              if(rq_write_lbl_request[index]):
                  if(is_ack(rq_comm_set_var("LBL", rq_write_lbl[index], socket))):
                      rq_write_lbl_previous[index] = rq_write_lbl[index]
                      rq_write_lbl_request[index] = False
                  end
              end

              if(rq_write_lgn_request[index]):
                  if(is_ack(rq_comm_set_var("LGN", rq_write_lgn[index], socket))):
                      rq_write_lgn_previous[index] = rq_write_lgn[index]
                      rq_write_lgn_request[index] = False
                  end
              end

              if(rq_write_msc_request[index]):
                  if(is_ack(rq_comm_set_var("MSC", rq_write_msc[index], socket))):
                      rq_write_msc_previous[index] = rq_write_msc[index]
                      rq_write_msc_request[index] = False
                  end
              end

              if(rq_write_mod_request[index]):
                  if(is_ack(rq_comm_set_var("MOD", rq_write_mod[index], socket))):
                      rq_write_mod_previous[index] = rq_write_mod[index]
                      rq_write_mod_request[index] = False
                  end
              end
          end
          index = index + 1
      end
  end

  def rq_activate(gripper_socket="1"):
      if (not rq_is_gripper_activated(gripper_socket)):
          rq_reset(gripper_socket)

          while(not rq_get_var("ACT", 1, gripper_socket) == 0 or not rq_get_var("STA", 1, gripper_socket) == 0):
              rq_reset(gripper_socket)
              sync()
          end

          rq_set_var("ACT",1, gripper_socket)
      end
  end

  def rq_activate_and_wait(gripper_socket="1"):
      if (not rq_is_gripper_activated(gripper_socket)):
          rq_activate(gripper_socket)
          sleep(1.0)

          while(not rq_get_var("ACT", 1, gripper_socket) == 1 or not rq_get_var("STA", 1, gripper_socket) == 3):
              sleep(0.1)
          end

          sleep(0.5)
      end
  end

  def rq_activate_all_grippers(reset=False):
      if(gripper_connected[0]):
          rq_reset_and_activate("1", reset)
      end

      if(gripper_connected[1]):
          rq_reset_and_activate("2", reset)
      end

      if(gripper_connected[2]):
          rq_reset_and_activate("3", reset)
      end

      if(gripper_connected[3]):
          rq_reset_and_activate("4", reset)
      end
  end

  def rq_reset_and_activate(gripper_socket="1", reset=False):
      if(reset):
          rq_reset(gripper_socket)
          rq_activate_and_wait(gripper_socket)
      elif(not rq_is_gripper_activated(gripper_socket)):
          rq_activate_and_wait(gripper_socket)
      end
  end

  def rq_reset(gripper_socket="1"):
      rq_set_var("ACT", 0, gripper_socket)
      rq_set_var("ATR", 0, gripper_socket)

      while(not rq_get_var("ACT", 1, gripper_socket) == 0 or not rq_get_var("STA", 1, gripper_socket) == 0):
          rq_set_var("ACT", 0, gripper_socket)
          rq_set_var("ATR", 0, gripper_socket)
          sync()
      end

      sleep(0.5)
  end

  def rq_auto_release_open_and_wait(gripper_socket="1"):
      rq_set_var("ATR",0, gripper_socket)
      rq_set_var("ARD",0, gripper_socket)
      rq_set_var("ACT",1, gripper_socket)
      sleep(0.1)
      rq_set_var("ATR",1, gripper_socket)

      rq_wait_autorelease_completed(gripper_socket)
  end

  def rq_auto_release_close_and_wait(gripper_socket="1"):
      rq_set_var("ATR",0, gripper_socket)
      rq_set_var("ARD",1, gripper_socket)
      rq_set_var("ACT",1, gripper_socket)
      sleep(0.1)
      rq_set_var("ATR",1, gripper_socket)

      rq_wait_autorelease_completed(gripper_socket)
  end

  def rq_wait_autorelease_completed(gripper_socket="1"):
      remainingRetries = 20
      gFLT = rq_get_var("FLT", 2, gripper_socket)

      while(not is_FLT_autorelease_in_progress(gFLT) and remainingRetries > 0):
          remainingRetries = remainingRetries - 1
          gFLT = rq_get_var("FLT", 2, gripper_socket)
          sleep(0.1)
      end

      remainingRetries = 100
      gFLT = rq_get_var("FLT", 2, gripper_socket)

      while(not is_FLT_autorelease_completed(gFLT) and remainingRetries > 0):
          remainingRetries = remainingRetries - 1
          gFLT = rq_get_var("FLT", 2, gripper_socket)
          sleep(0.1)
      end
  end

  def rq_set_force(force, gripper_socket="1"):
      force = floor(scale(force, [0, 255], [0.0, 255.0]))
      rq_set_var("FOR", force, gripper_socket)
  end

  def rq_set_speed(speed, gripper_socket="1"):
      speed = floor(scale(speed, [0, 255], [0.0, 255.0]))
      rq_set_var("SPE", speed, gripper_socket)
  end

  def rq_open(gripper_socket="1"):
      rq_move(0, gripper_socket)
  end

  def rq_close(gripper_socket="1"):
      rq_move(255, gripper_socket)
  end

  def rq_open_and_wait(gripper_socket="1"):
      rq_move_and_wait(0, gripper_socket)
  end

  def rq_close_and_wait(gripper_socket="1"):
      rq_move_and_wait(255, gripper_socket)
  end

  def rq_move(pos, gripper_socket="1"):
      rq_set_pos(pos, gripper_socket)
      rq_go_to(gripper_socket)
  end

  def rq_move_and_wait(pos, gripper_socket="1"):
      rq_move(pos, gripper_socket)

      while (not rq_is_motion_complete(gripper_socket)):
          # wait for motion completed
          sync()
      end
  end

  def rq_wait_for_pos_request(pos, gripper_socket="1"):
      gPRE = rq_get_var("PRE", 3, gripper_socket)

      while (gPRE != pos):
          rq_set_var("POS", pos, gripper_socket)
          sync()
          gPRE = rq_get_var("PRE", 3, gripper_socket)
      end
  end

  def rq_wait_pos_spe_for_request(pos, speed, force, gripper_socket="1"):
      gPRE = rq_get_var("PRE", 3, gripper_socket)

      while (gPRE != pos):
          rq_set_pos_spe_for_var(pos, speed, force, gripper_socket)
          sync()
          gPRE = rq_get_var("PRE", 3, gripper_socket)
      end
  end

  def rq_wait_for_pos(pos, gripper_socket="1"):
      rq_wait_for_pos_request(pos, gripper_socket)

      # Wait for the gripper motion to complete
      while (not rq_is_motion_complete(gripper_socket)):
          # wait for motion completed
          sync()
          rq_set_var("GTO", 1, gripper_socket)
      end
  end

  def rq_wait(gripper_socket="1"):
      # Wait for the gripper motion to complete
      while (not rq_is_motion_complete(gripper_socket)):
          sync()
          # The following patch is for Robotiq's Camera issue when communication is lost, but not the activation
          # the communication driver reset the GTO bit
          rq_set_var("GTO", 1, gripper_socket)
      end
  end

  def rq_wait_for_object_detected(gripper_socket="1"):
      # Wait the object detection
      while (not rq_is_object_detected(gripper_socket)):
          sync()
      end
  end

  # set the position
  def rq_set_pos(pos, gripper_socket="1"):
      pos = floor(scale(pos, [0, 255], [0.0, 255.0]))
      rq_set_var("POS", pos, gripper_socket)
      rq_wait_for_pos_request(pos, gripper_socket)
  end

  def rq_set_pos_spd_for(pos, speed, force, gripper_socket="1"):
      pos = floor(scale(pos, [0, 255], [0.0, 255.0]))
      speed = floor(scale(speed, [0, 255], [0.0, 255.0]))
      force = floor(scale(force, [0, 255], [0.0, 255.0]))

      rq_set_pos_spe_for_var(pos, speed, force, gripper_socket)
  end

  def rq_set_gripper_max_current_mA(current_mA, gripper_socket="1"):
      current = floor(current_mA / 10)

      rq_set_var("MSC", current, gripper_socket)
      current_read = rq_get_var("MSC", 1, gripper_socket)

      while(current_read != current):
          rq_set_var("MSC", current, gripper_socket)
          current_read = rq_get_var("MSC", 1, gripper_socket)
      end
  end

  def rq_set_gripper_mode(mode, gripper_socket="1"):
      rq_set_var("MOD", mode, gripper_socket)
  end

  def rq_set_gripper_max_cur(current_mA, gripper_socket="1"):
      rq_set_gripper_max_current_mA(current_mA, gripper_socket)
  end

  def rq_get_gripper_max_current_mA(gripper_socket="1"):
      current = rq_get_var("MSC", 1, gripper_socket)

      if(current == -1):
          current_mA = current
      else:
          current_mA = current * 10
      end

      return current_mA
  end

  def rq_get_gripper_max_cur(gripper_socket="1"):
      return rq_get_gripper_max_current_mA(gripper_socket)
  end

  def rq_set_max_current_for_all_grippers():
      current_mA = rq_get_max_current_mA()

      if(gripper_connected[0]):
          rq_set_gripper_max_current_mA(current_mA, "1")
      end

      if(gripper_connected[1]):
          rq_set_gripper_max_current_mA(current_mA, "2")
      end

      if(gripper_connected[2]):
          rq_set_gripper_max_current_mA(current_mA, "3")
      end

      if(gripper_connected[3]):
          rq_set_gripper_max_current_mA(current_mA, "4")
      end
  end

  def rq_get_max_current_mA():
      max_current_mA = 0

      if(rq_current_limit_enabled):
          nb_connected_grippers = rq_get_nb_connected_grippers()

          if(nb_connected_grippers == 1):
              max_current_mA = 600
          elif(nb_connected_grippers > 1):
              max_current_mA = 450
          end
      else:

      end

      return max_current_mA
  end

  def rq_get_nb_connected_grippers():
      nb_connected_grippers = 0

      if(gripper_connected[0]):
          nb_connected_grippers = nb_connected_grippers + 1
      end

      if(gripper_connected[1]):
          nb_connected_grippers = nb_connected_grippers + 1
      end

      if(gripper_connected[2]):
          nb_connected_grippers = nb_connected_grippers + 1
      end

      if(gripper_connected[3]):
          nb_connected_grippers = nb_connected_grippers + 1
      end

      return nb_connected_grippers
  end

  def rq_list_of_bytes_to_value(list_of_bytes):
      value = -1

      # response list length
      if (list_of_bytes[0] == 1):
          value = list_of_bytes[1] - 48
      elif (list_of_bytes[0] == 2):
          value = (list_of_bytes[1] - 48) * 10 + (list_of_bytes[2] - 48)
      elif (list_of_bytes[0] == 3):
          value = (list_of_bytes[1] - 48) * 100 + (list_of_bytes[2] - 48) * 10 + (list_of_bytes[3] - 48)
      end

      return value
  end

  def rq_is_motion_complete(gripper_socket="1"):
      gOBJ = rq_get_var("OBJ", 1, gripper_socket)
      sync()
      return is_OBJ_gripper_at_position(gOBJ) or is_OBJ_object_detected(gOBJ)
  end

  def rq_is_gripper_activated(gripper_socket="1"):
      gSTA = rq_get_var("STA", 1, gripper_socket)
      sync()
      return is_STA_gripper_activated(gSTA)
  end

  def rq_is_object_detected(gripper_socket="1"):
      gOBJ = rq_get_var("OBJ", 1, gripper_socket)
      sync()
      return is_OBJ_object_detected(gOBJ)
  end

  def rq_current_pos(gripper_socket="1"):
      gPOS = rq_get_var("POS", 1, gripper_socket)
      sync()
      return gPOS
  end

  def rq_motor_current(gripper_socket="1"):
      rq_current = rq_get_var("COU", 1, gripper_socket)
      sync()
      return rq_current * 10
  end

  def rq_print_connected_grippers():
      if(gripper_connected[0]):
          textmsg("Gripper 1 : ", "connected and socket open.")
      end

      if (gripper_connected[1]):
          textmsg("Gripper 2 : ", "connected and socket open.")
      end

      if (gripper_connected[2]):
          textmsg("Gripper 3 : ", "connected and socket open.")
      end

      if (gripper_connected[3]):
          textmsg("Gripper 4 : ", "connected and socket open.")
      end
  end

  def rq_print_gripper_fault_code(gripper_socket="1"):
      gFLT = rq_get_var("FLT", 2, gripper_socket)

      if(is_FLT_no_fault(gFLT)):
          textmsg("Gripper Fault : ", "No Fault (0x00)")
      elif (is_FLT_action_delayed(gFLT)):
          textmsg("Gripper Fault : ", "Priority Fault: Action delayed, initialization must be completed prior to action (0x05)")
      elif (is_FLT_not_activated(gFLT)):
          textmsg("Gripper Fault : ", "Priority Fault: The activation must be set prior to action (0x07)")
      elif (is_FLT_autorelease_in_progress(gFLT)):
          textmsg("Gripper Fault : ", "Minor Fault: Automatic release in progress (0x0B)")
      elif (is_FLT_overcurrent(gFLT)):
          textmsg("Gripper Fault : ", "Minor Fault: Overcurrent protection triggered (0x0E)")
      elif (is_FLT_autorelease_completed(gFLT)):
          textmsg("Gripper Fault : ", "Major Fault: Automatic release completed (0x0F)")
      else:
          textmsg("Gripper Fault : ", "Unknown Fault")
      end
  end

  def rq_print_gripper_num_cycles(gripper_socket="1"):
      num_cycles = rq_get_var("NCY", 1, gripper_socket)

      if(num_cycles == -1):
          textmsg("Gripper Cycle Number : ", "Number of cycles is unreachable.")
      else:
          textmsg("Gripper Cycle Number : ", num_cycles)
      end
  end

  def rq_print_gripper_driver_state(gripper_socket="1"):
      driver_state = rq_get_var("DST", 1, gripper_socket)

      if(driver_state == 0):
          textmsg("Gripper Driver State : ", "RQ_STATE_INIT")
      elif(driver_state == 1):
          textmsg("Gripper Driver State : ", "RQ_STATE_LISTEN")
      elif(driver_state == 2):
          textmsg("Gripper Driver State : ", "RQ_STATE_READ_INFO")
      elif(driver_state == 3):
          textmsg("Gripper Driver State : ", "RQ_STATE_ACTIVATION")
      else:
          textmsg("Gripper Driver State : ", "RQ_STATE_RUN")
      end
  end

  def rq_print_gripper_serial_number(gripper_socket="1"):
      serial_number = rq_get_var_string("SNU", 1, gripper_socket)
      textmsg("Gripper Serial Number : ", serial_number)
  end

  def rq_print_gripper_firmware_version(gripper_socket="1"):
      firmware_version = rq_get_var_string("FWV", 1, gripper_socket)
      textmsg("Gripper Firmware Version : ", firmware_version)
  end

  def rq_print_gripper_driver_version(gripper_socket="1"):
      driver_version = rq_get_var_string("VER", 1, gripper_socket)
      textmsg("Gripper Driver Version : ", driver_version)
  end

  def rq_print_gripper_connection_state(gripper_socket="1"):
      connection_state = rq_get_var("PCO", 1, gripper_socket)

      if (connection_state == 0):
          textmsg("Gripper Connection State : ", "No connection problem detected")
      else:
          textmsg("Gripper Connection State : ", "Connection problem detected")
      end
  end

  # Returns True if list_of_bytes is [3, 'a', 'c', 'k']
  def is_ack(list_of_bytes):

      # list length is not 3
      if (list_of_bytes[0] != 3):
          return False
      end

      # first byte not is 'a'?
      if (list_of_bytes[1] != 97):
          return False
      end

      # first byte not is 'c'?
      if (list_of_bytes[2] != 99):
          return False
      end

      # first byte not is 'k'?
      if (list_of_bytes[3] != 107):
          return False
      end

      return True
  end

  # Returns True if list_of_bytes is not [3, 'a', 'c', 'k']
  def is_not_ack(list_of_bytes):
      if (is_ack(list_of_bytes)):
          return False
      else:
          return True
      end
  end

  def is_STA_gripper_activated (gSTA):
      if (gSTA == 3):
          return True
      end

      return False
  end

  def is_OBJ_object_detected (gOBJ):
      if (gOBJ == 1 or gOBJ == 2):
          return True
      end

      return False
  end

  def is_OBJ_gripper_at_position (gOBJ):
      if (gOBJ == 3):
          return True
      end

      return False
  end

  def is_not_OBJ_gripper_at_position (gOBJ):
      if (is_OBJ_gripper_at_position(gOBJ)):
          return False
      else:
          return True
      end
  end

  #### GTO Section ####
  def rq_stop(gripper_socket="1"):
      rq_set_var("GTO", 0, gripper_socket)
  end

  def rq_set_GTO_and_wait(value, gripper_socket="1"):
      rq_set_var("GTO" ,value, gripper_socket)
      while(not is_GTO(value, rq_get_var("GTO", 1, gripper_socket))):
        sync()
      end
  end

  def rq_go_to(gripper_socket="1"):
      rq_set_var("GTO", 1, gripper_socket)
  end


  def is_GTO(goto_value, rGTO):
      return rGTO == goto_value
  end
  #### GTO Section ####

  def is_FLT_no_fault(gFLT):
      return gFLT == 0
  end

  def is_FLT_warning(gFLT):
      return gFLT >= 1 and gFLT <= 7
  end

  def is_FLT_faulted(gFLT):
      return gFLT >= 8
  end

  def is_FLT_action_delayed(gFLT):
      return gFLT == 5
  end

  def is_FLT_not_activated(gFLT):
      return gFLT == 7
  end

  def is_FLT_autorelease_in_progress(gFLT):
      return gFLT == 11
  end

  def is_FLT_overcurrent(gFLT):
      return gFLT == 14
  end

  def is_FLT_autorelease_completed(gFLT):
      return gFLT == 15
  end

  def rq_set_var(var_name, var_value, gripper_socket="1"):
      index = rq_socket_to_index(gripper_socket)

      enter_critical

      if (var_name == "ACT"):
          rq_write_act[index] = var_value
          rq_write_act_request[index] = True
      elif (var_name == "GTO"):
          rq_write_gto[index] = var_value
          rq_write_gto_request[index] = True
      elif (var_name == "ATR"):
          rq_write_atr[index] = var_value
          rq_write_atr_request[index] = True
      elif (var_name == "ARD"):
          rq_write_ard[index] = var_value
          rq_write_ard_request[index] = True
      elif (var_name == "FOR"):
          rq_write_for[index] = var_value
          rq_write_pos_request[index] = True
      elif (var_name == "SPE"):
          rq_write_spe[index] = var_value
          rq_write_pos_request[index] = True
      elif (var_name == "POS"):
          rq_write_pos[index] = var_value
          rq_write_pos_request[index] = True
      elif (var_name == "LBP"):
          rq_write_lbp[index] = var_value
          rq_write_lbp_request[index] = True
      elif (var_name == "LRD"):
          rq_write_lrd[index] = var_value
          rq_write_lrd_request[index] = True
      elif (var_name == "LBL"):
          rq_write_lbl[index] = var_value
          rq_write_lbl_request[index] = True
      elif (var_name == "LGN"):
          rq_write_lgn[index] = var_value
          rq_write_lgn_request[index] = True
      elif (var_name == "MSC"):
          rq_write_msc[index] = var_value
          rq_write_msc_request[index] = True
      elif (var_name == "MOD"):
          rq_write_mod[index] = var_value
          rq_write_mod_request[index] = True
      end

      exit_critical

      if (var_name == "ACT"):
          while(rq_write_act_request[index]):
              sync()
          end
      elif (var_name == "GTO"):
          while(rq_write_gto_request[index]):
              sync()
          end
      elif (var_name == "ATR"):
          while(rq_write_atr_request[index]):
              sync()
          end
      elif (var_name == "ARD"):
          while(rq_write_ard_request[index]):
              sync()
          end
      elif (var_name == "FOR"):
          while(rq_write_pos_request[index]):
              sync()
          end
      elif (var_name == "SPE"):
          while(rq_write_pos_request[index]):
              sync()
          end
      elif (var_name == "POS"):
          while(rq_write_pos_request[index]):
              sync()
          end
      elif (var_name == "LBP"):
          while(rq_write_lbp_request[index]):
              sync()
          end
      elif (var_name == "LRD"):
          while(rq_write_lrd_request[index]):
              sync()
          end
      elif (var_name == "LBL"):
          while(rq_write_lbl_request[index]):
              sync()
          end
      elif (var_name == "LGN"):
          while(rq_write_lgn_request[index]):
              sync()
          end
      elif (var_name == "MSC"):
          while(rq_write_msc_request[index]):
              sync()
          end
      elif (var_name == "MOD"):
          while(rq_write_mod_request[index]):
              sync()
          end
      end
  end

  def rq_set_pos_spe_for_var(pos, speed, force, gripper_socket="1"):
      index = rq_socket_to_index(gripper_socket)

      enter_critical

      rq_write_for[index] = force
      rq_write_spe[index] = speed
      rq_write_pos[index] = pos
      rq_write_pos_request[index] = True

      exit_critical
  end

  def rq_get_var(var_name, nbr_bytes, gripper_socket="1"):
      index = rq_socket_to_index(gripper_socket)
      var_value = -1

      if (var_name == "ACT"):
          enter_critical
          rq_read_act_req[index] = True
          exit_critical
          while(rq_read_act_req[index]):
              sync()
          end
          var_value = rq_read_act[index]

      elif (var_name == "GTO"):
          enter_critical
          rq_read_gto_req[index] = True
          exit_critical
          while(rq_read_gto_req[index]):
              sync()
          end
          var_value = rq_read_gto[index]

      elif (var_name == "FOR"):
          enter_critical
          rq_read_for_req[index] = True
          exit_critical
          while(rq_read_for_req[index]):
              sync()
          end
          var_value = rq_read_for[index]

      elif (var_name == "SPE"):
          enter_critical
          rq_read_spe_req[index] = True
          exit_critical
          while(rq_read_spe_req[index]):
              sync()
          end
          var_value = rq_read_spe[index]

      elif (var_name == "OBJ"):
          enter_critical
          rq_read_obj_req[index] = True
          exit_critical
          while(rq_read_obj_req[index]):
              sync()
          end
          var_value = rq_read_obj[index]

      elif (var_name == "STA"):
          enter_critical
          rq_read_sta_req[index] = True
          exit_critical
          while(rq_read_sta_req[index]):
              sync()
          end
          var_value = rq_read_sta[index]

      elif (var_name == "FLT"):
          enter_critical
          rq_read_flt_req[index] = True
          exit_critical
          while(rq_read_flt_req[index]):
              sync()
          end
          var_value = rq_read_flt[index]

      elif (var_name == "POS"):
          enter_critical
          rq_read_pos_req[index] = True
          exit_critical
          while(rq_read_pos_req[index]):
              sync()
          end
          var_value = rq_read_pos[index]

      elif (var_name == "PRE"):
          enter_critical
          rq_read_pre_req[index] = True
          exit_critical
          while(rq_read_pre_req[index]):
              sync()
          end
          var_value = rq_read_pre[index]

      elif (var_name == "LBP"):
          enter_critical
          rq_read_lbp_req[index] = True
          exit_critical
          while(rq_read_lbp_req[index]):
              sync()
          end
          var_value = rq_read_lbp[index]

      elif (var_name == "LRD"):
          enter_critical
          rq_read_lrd_req[index] = True
          exit_critical
          while(rq_read_lrd_req[index]):
              sync()
          end
          var_value = rq_read_lrd[index]

      elif (var_name == "LBL"):
          enter_critical
          rq_read_lbl_req[index] = True
          exit_critical
          while(rq_read_lbl_req[index]):
              sync()
          end
          var_value = rq_read_lbl[index]

      elif (var_name == "LGN"):
          enter_critical
          rq_read_lgn_req[index] = True
          exit_critical
          while(rq_read_lgn_req[index]):
              sync()
          end
          var_value = rq_read_lgn[index]

      elif (var_name == "MSC"):
          enter_critical
          rq_read_msc_req[index] = True
          exit_critical
          while(rq_read_msc_req[index]):
              sync()
          end
          var_value = rq_read_msc[index]

      elif (var_name == "MOD"):
          enter_critical
          rq_read_mod_req[index] = True
          exit_critical
          while(rq_read_mod_req[index]):
              sync()
          end
          var_value = rq_read_mod[index]

      elif (var_name == "NCY"):
          enter_critical
          rq_read_ncy_req[index] = True
          exit_critical
          while(rq_read_ncy_req[index]):
              sync()
          end
          var_value = rq_read_ncy[index]

      elif (var_name == "PCO"):
          enter_critical
          rq_read_pco_req[index] = True
          exit_critical
          while(rq_read_pco_req[index]):
              sync()
          end
          var_value = rq_read_pco[index]

      elif (var_name == "DST"):
          enter_critical
          rq_read_dst_req[index] = True
          exit_critical
          while(rq_read_dst_req[index]):
              sync()
          end
          var_value = rq_read_dst[index]

      end

      return var_value
  end

  def rq_get_var_string(var_name, nbr_bytes, gripper_socket="1"):
      index = rq_socket_to_index(gripper_socket)
      var_value = ""

      enter_critical

      if (var_name == "SNU"):
          if(gripper_socket == "1"):
              var_value = rq_read_snu_1
          elif(gripper_socket == "2"):
              var_value = rq_read_snu_2
          elif(gripper_socket == "3"):
              var_value = rq_read_snu_3
          elif(gripper_socket == "4"):
              var_value = rq_read_snu_4
          end
      elif (var_name == "FWV"):
          if(gripper_socket == "1"):
              var_value = rq_read_fwv_1
          elif(gripper_socket == "2"):
              var_value = rq_read_fwv_2
          elif(gripper_socket == "3"):
              var_value = rq_read_fwv_3
          elif(gripper_socket == "4"):
              var_value = rq_read_fwv_4
          end
      elif (var_name == "VER"):
          if(gripper_socket == "1"):
              var_value = rq_read_ver_1
          elif(gripper_socket == "2"):
              var_value = rq_read_ver_2
          elif(gripper_socket == "3"):
              var_value = rq_read_ver_3
          elif(gripper_socket == "4"):
              var_value = rq_read_ver_4
          end
      end

      exit_critical

      return var_value
  end

  def rq_is_object_validated(gripper_selected, gripper_socket="1"):
      if(gripper_selected):
          if(rq_is_object_detected(gripper_socket)):
              return True
          else:
              return False
          end
      else:
          return True
      end
  end

  ############################################
  # normalized functions (maps 0-100 to 0-255)
  ############################################
  def rq_set_force_norm(force_norm, gripper_socket="1"):
      force_gripper = norm_to_gripper(force_norm)
      rq_set_force(force_gripper, gripper_socket)
  end

  def rq_set_speed_norm(speed_norm, gripper_socket="1"):
      speed_gripper = norm_to_gripper(speed_norm)
      rq_set_speed(speed_gripper, gripper_socket)
  end

  def rq_move_norm(pos_norm, gripper_socket="1"):
      pos_gripper = norm_to_gripper(pos_norm)
      rq_move(pos_gripper, gripper_socket)
  end

  def rq_move_and_wait_norm(pos_norm, gripper_socket="1"):
      pos_gripper = norm_to_gripper(pos_norm)
      rq_move_and_wait(pos_gripper, gripper_socket)
  end

  def rq_set_pos_norm(pos_norm, gripper_socket="1"):
      pos_gripper = norm_to_gripper(pos_norm)
      rq_set_pos(pos_gripper, gripper_socket)
  end

  def rq_current_pos_norm(gripper_socket="1"):
      pos_gripper = rq_current_pos(gripper_socket)
      pos_norm = gripper_to_norm(pos_gripper)
      return pos_norm
  end

  def gripper_to_norm(value_gripper):
      value_norm = (value_gripper / 255) * 100
      return floor(value_norm)
  end

  def norm_to_gripper(value_norm):
      value_gripper = (value_norm / 100) * 255
      return ceil(value_gripper)
  end

  def rq_get_position():
      return rq_current_pos_norm()
  end

  def rq_gripper_led_on(gripper_socket="1"):
      rq_set_var("LBP",0, gripper_socket)
  end

  def rq_gripper_led_off(gripper_socket="1"):
      rq_set_var("LBP",1, gripper_socket)
      rq_set_var("LRD",0, gripper_socket)
      rq_set_var("LBL",0, gripper_socket)
      rq_set_var("LGN",0, gripper_socket)
  end

  def rq_gripper_led_force_red(gripper_socket="1"):
      rq_set_var("LBP",1, gripper_socket)
      rq_set_var("LRD",1, gripper_socket)
      rq_set_var("LBL",0, gripper_socket)
      rq_set_var("LGN",0, gripper_socket)
  end

  def rq_gripper_led_force_blue(gripper_socket="1"):
      rq_set_var("LBP",1, gripper_socket)
      rq_set_var("LRD",0, gripper_socket)
      rq_set_var("LBL",1, gripper_socket)
      rq_set_var("LGN",0, gripper_socket)
  end

  def rq_gripper_led_force_green(gripper_socket="1"):
      rq_set_var("LBP",1, gripper_socket)
      rq_set_var("LRD",0, gripper_socket)
      rq_set_var("LBL",0, gripper_socket)
      rq_set_var("LGN",1, gripper_socket)
  end

  def rq_gripper_led_force_purple(gripper_socket="1"):
      rq_set_var("LBP",1, gripper_socket)
      rq_set_var("LRD",1, gripper_socket)
      rq_set_var("LBL",1, gripper_socket)
      rq_set_var("LGN",0, gripper_socket)
  end

  ############################################
  # mm/inches functions
  ############################################
  gripper_closed_norm = [100, 100, 100, 100]
  gripper_open_norm = [0, 0, 0, 0]
  gripper_closed_mm = [0, 0, 0, 0]
  gripper_open_mm = [50, 50, 50, 50]

  def rq_current_pos_mm(gripper_socket=1):
      pos_gripper = rq_current_pos(gripper_socket)
      pos_mm = gripper_to_mm(pos_gripper, gripper_socket)
      return round_value_2_dec(pos_mm)
  end

  def rq_current_pos_inches(gripper_socket=1):
      pos_gripper = rq_current_pos(gripper_socket)
      pos_mm = gripper_to_mm(pos_gripper, gripper_socket)
      pos_in = pos_mm / 25.4
      return round_value_2_dec(pos_in)
  end

  def rq_move_mm(pos_mm, gripper_socket=1):
      pos_gripper = mm_to_gripper(pos_mm, gripper_socket)
      rq_move(pos_gripper, gripper_socket)
  end

  def rq_move_and_wait_mm(pos_mm, gripper_socket=1):
      pos_gripper = mm_to_gripper(pos_mm, gripper_socket)
      rq_move_and_wait(pos_gripper, gripper_socket)
  end

  def rq_move_inches(pos_in, gripper_socket=1):
      pos_mm = pos_in * 25.4
      rq_move_mm(pos_mm, gripper_socket)
  end

  def rq_move_and_wait_inches(pos_in, gripper_socket=1):
      pos_mm = pos_in * 25.4
      rq_move_and_wait_mm(pos_mm, gripper_socket)
  end

  def get_closed_norm(gripper_socket):
      return gripper_closed_norm[gripper_socket - 1]
  end

  def get_open_norm(gripper_socket):
      return gripper_open_norm[gripper_socket - 1]
  end

  def get_closed_mm(gripper_socket):
      return gripper_closed_mm[gripper_socket - 1]
  end

  def get_open_mm(gripper_socket):
      return gripper_open_mm[gripper_socket - 1]
  end

  def set_closed_norm(closed_norm, gripper_socket):
      gripper_closed_norm[gripper_socket - 1] = closed_norm
  end

  def set_open_norm(open_norm, gripper_socket):
      gripper_open_norm[gripper_socket - 1] = open_norm
  end

  def set_closed_mm(closed_mm, gripper_socket):
      gripper_closed_mm[gripper_socket - 1] = closed_mm
  end

  def set_open_mm(open_mm, gripper_socket):
      gripper_open_mm[gripper_socket - 1] = open_mm
  end

  def gripper_to_mm(value_gripper, gripper_socket):
      closed_norm = get_closed_norm(gripper_socket)
      open_norm = get_open_norm(gripper_socket)
      closed_mm = get_closed_mm(gripper_socket)
      open_mm = get_open_mm(gripper_socket)

      value_norm = (value_gripper / 255) * 100

      slope = (closed_mm - open_mm) / (closed_norm - open_norm)
      value_mm = slope * (value_norm - closed_norm) + closed_mm

      if (value_mm > open_mm):
          value_mm_limited = open_mm
      elif (value_mm < closed_mm):
          value_mm_limited = closed_mm
      else:
          value_mm_limited = value_mm
      end

      return value_mm_limited
  end

  def mm_to_gripper(value_mm, gripper_socket):
      closed_norm = get_closed_norm(gripper_socket)
      open_norm = get_open_norm(gripper_socket)
      closed_mm = get_closed_mm(gripper_socket)
      open_mm = get_open_mm(gripper_socket)

      slope = (closed_norm - open_norm) / (closed_mm - open_mm)
      value_norm = (value_mm - closed_mm) * slope + closed_norm

      value_gripper = value_norm * 255 / 100

      if (value_gripper > 255):
          value_gripper_limited = 255
      elif (value_gripper < 0):
          value_gripper_limited = 0
      else:
          value_gripper_limited = round_value(value_gripper)
      end

      return value_gripper_limited
  end

  def round_value(value):
      value_mod = value % 1

      if(value_mod < 0.5):
          return floor(value)
      else:
          return ceil(value)
      end
  end

  def round_value_2_dec(value):
      value_x_100 = value * 100
      value_x_100_rounded = round_value(value_x_100)
      return value_x_100_rounded / 100
  end

  def clear_socket_buffer(gripper_socket="1", read_timeout = 0.1):
      rq_comm_clear_socket_buffer_enabled[rq_socket_to_index(gripper_socket)] = True
  end

  def rq_gripper_id_to_ascii(gripper_id):
      if(gripper_id == "1"):
          return 57
      elif(gripper_id == "2"):
          return 50
      elif(gripper_id == "3"):
          return 51
      elif(gripper_id == "4"):
          return 52
      end
  end

  def scale(value, rawRange, scaledRange):
      def computeSlope(inputRange, outputRange):
          outputRangeDelta = outputRange[1] - outputRange[0]
          inputRangeDelta = inputRange[1] - inputRange[0]

          if (inputRangeDelta == 0):
              return 0
          else:
              return outputRangeDelta / inputRangeDelta
          end
      end

      def computeIntercept(slope, inputRange, outputRange):
          return outputRange[0] - (slope * inputRange[0])
      end

      def clipScaledValue(outputScaledValue, outputRange):
          if (outputRange[0] < outputRange[1]):
              return clipWhenLowerLimitIsLessThanHigher(outputScaledValue, outputRange)
          else:
              return clipWhenLowerLimitIsGreaterThanHigherLimit(outputScaledValue, outputRange)
          end
      end

      def clipWhenLowerLimitIsGreaterThanHigherLimit(outputScaledValue, outputRange):
          if (outputScaledValue < outputRange[1]):
              return outputRange[1]
          elif (outputScaledValue > outputRange[0]):
              return outputRange[0]
          else:
              return outputScaledValue
          end
      end

      def clipWhenLowerLimitIsLessThanHigher(outputScaledValue, outputRange):
          if (outputScaledValue < outputRange[0]):
              return outputRange[0]
          elif (outputScaledValue > outputRange[1]):
              return outputRange[1]
          else:
              return outputScaledValue
          end
      end

      slope = computeSlope(rawRange, scaledRange)
      intercept = computeIntercept(slope, rawRange, scaledRange)
      scaledValue = slope * value + intercept
      return clipScaledValue(scaledValue, scaledRange)
  end

  def limit(value, range):
      return scale(value, range, range)
  end


  rq_init_comm_if_connected(9, "1")
  rq_init_comm_if_connected(2, "2")
  rq_init_comm_if_connected(3, "3")
  rq_init_comm_if_connected(4, "4")
  rq_print_connected_grippers()
  rq_gripper_communication_thread = run rq_gripper_communication()
  set_closed_norm(100.0, 1)
  set_open_norm(0.0, 1)
  set_closed_mm(0.0, 1)
  set_open_mm(50.0, 1)
  set_closed_norm(100.0, 2)
  set_open_norm(0.0, 2)
  set_closed_mm(0.0, 2)
  set_open_mm(50.0, 2)
  set_closed_norm(100.0, 3)
  set_open_norm(0.0, 3)
  set_closed_mm(0.0, 3)
  set_open_mm(50.0, 3)
  set_closed_norm(100.0, 4)
  set_open_norm(0.0, 4)
  set_closed_mm(0.0, 4)
  set_open_mm(50.0, 4)
  rq_current_limit_enabled = False
  while(not rq_gripper_communication_thread_started):
      sync()
  end
  # end: URCap Installation Node
  global Waypoint_13_p=p[.463075378858, -.033118898203, .367768326041, -2.244549547112, 2.186980266689, -.146698143579]
  global Waypoint_13_q=[0.2635507583618164, -1.4171207708171387, -1.6266908645629883, -1.6176563702025355, 1.4933080673217773, 0.2373518943786621]
  global Waypoint_4_p=p[.590056785195, .345400457164, .346404902266, -2.196998113937, 2.219440293840, -.040291679599]
  global Waypoint_4_q=[0.7344789505004883, -1.997808118859762, -1.0045957565307617, -1.6909080944456996, 1.5455546379089355, 0.7456479072570801]
  global Waypoint_14_p=p[.590691955827, .347823211240, .305526547873, 2.172764276997, -2.166287134815, .069902761340]
  global Waypoint_14_q=[0.7456297874450684, -2.05458464244985, -1.0044755935668945, -1.724589010278219, 1.5220775604248047, 0.7456116676330566]
  global Waypoint_6_p=p[.590703087407, .382182873249, .328360235165, 1.950028721832, -1.951627591374, .449966499654]
  global Waypoint_6_q=[0.8704757690429688, -2.380897661248678, -0.39194202423095703, -2.3245274029173792, 1.2879180908203125, 0.9274992942810059]
  global Waypoint_01_p=p[.571574269346, .374397712413, .371422124647, 1.961688310974, -2.391957405826, .029489865356]
  global Waypoint_01_q=[0.7810592651367188, -2.0693794689574183, -0.815150260925293, -1.8778792820372523, 1.5559697151184082, 0.979529857635498]
  global Waypoint_001_p=p[.493332912072, .240993851770, .371404564950, 1.961666742853, -2.391915578890, .029514935952]
  global Waypoint_001_q=[0.7068662643432617, -1.7017342052855433, -1.3084897994995117, -1.7510363064207972, 1.5530376434326172, 0.9058690071105957]
  global Waypoint_02_p=p[.526745143140, .237719312996, .291293390808, 1.950208204135, -2.458073573808, .012375221811]
  global Waypoint_02_q=[0.6587648391723633, -1.7409912548460902, -1.4781064987182617, -1.4974926275065918, 1.5630850791931152, 0.889859676361084]
  global Waypoint_03_p=p[.526751742730, .350284344668, .291328413416, 1.950187440714, -2.458204313759, .012252654607]
  global Waypoint_03_q=[0.8008732795715332, -1.875624795953268, -1.308670997619629, -1.5332802099040528, 1.5635037422180176, 1.0318779945373535]
  global Waypoint_11_p=p[.463069913685, .373635307885, .367778231425, -2.552402103854, 1.792810489584, -.143117491211]
  global Waypoint_11_q=[0.9444355964660645, -1.758153577844137, -1.2712469100952148, -1.6630522213377894, 1.479501724243164, 0.5989480018615723]
  global Waypoint_04_p=p[.454818817763, .411321007042, .329882546598, -2.306666213389, 2.117267733564, -.146324640661]
  global Waypoint_04_q=[0.9934988021850586, -1.8158890209593714, -1.2895774841308594, -1.6158977947630824, 1.4775753021240234, 0.9098916053771973]
  global Waypoint_05_p=p[.454825579913, .411325549870, .275128730836, -2.306691410841, 2.117311031571, -.146386460588]
  global Waypoint_05_q=[0.9934391975402832, -1.8203073940672816, -1.4238080978393555, -1.47730906427417, 1.477550983428955, 0.9099392890930176]
  global Waypoint_06_p=p[.454819389507, .411334060077, .291839713142, -2.306690216015, 2.117222333267, -.146333888287]
  global Waypoint_06_q=[0.9934630393981934, -1.817026277581686, -1.3852167129516602, -1.5191114705852051, 1.4775753021240234, 0.9098916053771973]
  $ 1 "BeforeStart"
  $ 2 "MoveJ"
  $ 3 "Waypoint_13" "breakAfter"
  movej(get_inverse_kin(Waypoint_13_p, qnear=Waypoint_13_q), a=1.3962634015954636, v=1.0471975511965976)
  # begin: URCap Program Node
  #   Source: Robotiq_Grippers, 1.8.3.4198-beta, Robotiq Inc.
  #   Type: Gripper Activate
  $ 4 "Gripper Activate"

  kill rq_gripper_communication_thread
  rq_gripper_communication_thread_started = False

  rq_init_comm_if_connected(9, "1")
  rq_init_comm_if_connected(2, "2")
  rq_init_comm_if_connected(3, "3")
  rq_init_comm_if_connected(4, "4")
  rq_print_connected_grippers()
  rq_gripper_communication_thread = run rq_gripper_communication()

  while(not rq_gripper_communication_thread_started):
      sync()
  end

  rq_set_max_current_for_all_grippers()

  reset_and_activate = False

  rq_activate_all_grippers(False)
  # end: URCap Program Node
  $ 5 "If  not digital_in[4]"
  if (  not  get_standard_digital_in(4)):
    $ 6 "Popup: Postavi skatlo k zadnjemu senzorju :)"
    popup("Postavi skatlo k zadnjemu senzorju :)", "Message", False, False, blocking=True)
    $ 7 "Loop  not digital_in[4]"
    while (  not  get_standard_digital_in(4)):
      $ 8 "'prazen loop ne laufa :)'"
      # 'prazen loop ne laufa :)'
      $ 9 "Wait: 0.01"
      sleep(0.01)
    end
  end
  $ 10 "open_socket≔socket_open('192.168.65.102',50000,'student')"
  global open_socket=socket_open("192.168.65.102",50000,"student")
  $ 11 "Loop  not open_socket"
  while (  not  open_socket):
    $ 12 "open_socket≔socket_open('192.168.65.102',50000,'student')"
    global open_socket=socket_open("192.168.65.102",50000,"student")
  end
  $ 13 "Robot Program"
  $ 14 "MoveL"
  $ 15 "Waypoint_4" "breakAfter"
  movel(Waypoint_4_p, a=1.2, v=0.25)
  # begin: URCap Program Node
  #   Source: Robotiq_Grippers, 1.8.3.4198-beta, Robotiq Inc.
  #   Type: Gripper
  $ 16 "Gripper Open (2)"
  if not(gripper_connected[1]):
    popup("Gripper 2 must be connected to run this program.", "No connection", False, True, True)
  end
  if not(rq_is_gripper_activated("2")):
    popup("Gripper 2 is not activated. Go to Installation tab > Gripper to activate it and run the program again.", "Not activated", False, True, True)
  end
  rq_set_pos_spd_for(0, 0, 0, "2")
  rq_wait_pos_spe_for_request(0, 0, 0, "2")
  rq_go_to("2")
  rq_wait("2")
  # end: URCap Program Node
  $ 17 "If  not digital_in[5]"
  if (  not  get_standard_digital_in(5)):
    $ 18 "Set DO[5]=On"
    set_standard_digital_out(5, True)
  end
  $ 19 "Loop  not digital_in[5]"
  while (  not  get_standard_digital_in(5)):
    $ 20 "'cakam da se skatla pripelje'"
    # 'cakam da se skatla pripelje'
    $ 21 "Wait: 0.01"
    sleep(0.01)
  end
  $ 22 "Set DO[5]=Off"
  set_standard_digital_out(5, False)
  $ 23 "'tcp ip skatla prispela'"
  # 'tcp ip skatla prispela'
  $ 24 "If open_socket"
  if (open_socket):
    $ 25 "was_send≔socket_send_string('PRISPELA','student')"
    global was_send=socket_send_string("PRISPELA","student")
    $ 26 "Loop  not was_send"
    while (  not  was_send):
      $ 27 "was_send≔socket_send_string('PRISPELA','student')"
      global was_send=socket_send_string("PRISPELA","student")
      $ 28 "Wait: 0.01"
      sleep(0.01)
    end
    $ 29 "Wait: 0.01"
    sleep(0.01)
  end
  $ 30 "MoveL"
  $ 31 "Waypoint_14" "breakAfter"
  movel(Waypoint_14_p, a=1.2, v=0.25)
  $ 32 "'premik za prijem pokrova'"
  # 'premik za prijem pokrova'
  $ 33 "Set DO[0]=On"
  set_standard_digital_out(0, True)
  $ 34 "'vkopi napajanje za kljucavnico'"
  # 'vkopi napajanje za kljucavnico'
  $ 35 "Wait: 1.0"
  sleep(1.0)
  $ 36 "Set DO[0]=Off"
  set_standard_digital_out(0, False)
  # begin: URCap Program Node
  #   Source: Robotiq_Grippers, 1.8.3.4198-beta, Robotiq Inc.
  #   Type: Gripper
  $ 37 "Gripper Close (2)"
  if not(gripper_connected[1]):
    popup("Gripper 2 must be connected to run this program.", "No connection", False, True, True)
  end
  if not(rq_is_gripper_activated("2")):
    popup("Gripper 2 is not activated. Go to Installation tab > Gripper to activate it and run the program again.", "Not activated", False, True, True)
  end
  rq_set_pos_spd_for(255, 0, 71, "2")
  rq_wait_pos_spe_for_request(255, 0, 71, "2")
  rq_go_to("2")
  rq_wait("2")
  # end: URCap Program Node
  $ 38 "'gripper primer pokrov'"
  # 'gripper primer pokrov'
  $ 39 "'tcp ip skatla odklenjena'"
  # 'tcp ip skatla odklenjena'
  $ 40 "If open_socket"
  if (open_socket):
    $ 41 "was_send≔socket_send_string('ODKLENJENA','student')"
    global was_send=socket_send_string("ODKLENJENA","student")
    $ 42 "Loop  not was_send"
    while (  not  was_send):
      $ 43 "was_send≔socket_send_string('ODKLENJENA','student')"
      global was_send=socket_send_string("ODKLENJENA","student")
      $ 44 "Wait: 0.01"
      sleep(0.01)
    end
    $ 45 "Wait: 0.01"
    sleep(0.01)
  end
  $ 49 "'tcp_ip skatla je odprta'"
  # 'tcp_ip skatla je odprta'
  $ 50 "If open_socket"
  if (open_socket):
    $ 51 "was_send≔socket_send_string('ODPRTA','student')"
    global was_send=socket_send_string("ODPRTA","student")
    $ 52 "Loop  not was_send"
    while (  not  was_send):
      $ 53 "was_send≔socket_send_string('ODPRTA','student')"
      global was_send=socket_send_string("ODPRTA","student")
      $ 54 "Wait: 0.01"
      sleep(0.01)
    end
    $ 55 "Wait: 0.01"
    sleep(0.01)
  end
  $ 56 "'izklopi napajanje kljucavice (<4s)'"
  # 'izklopi napajanje kljucavice (<4s)'
  $ 57 "MoveL"
  $ 58 "Waypoint_6" "breakAfter"
  movel(Waypoint_6_p, a=1.2, v=0.25)
  $ 59 "'pokrov premakne blizje zadnjemu delu skatle'"
  # 'pokrov premakne blizje zadnjemu delu skatle'
  # begin: URCap Program Node
  #   Source: Robotiq_Grippers, 1.8.3.4198-beta, Robotiq Inc.
  #   Type: Gripper
  $ 60 "Gripper Open (2)"
  if not(gripper_connected[1]):
    popup("Gripper 2 must be connected to run this program.", "No connection", False, True, True)
  end
  if not(rq_is_gripper_activated("2")):
    popup("Gripper 2 is not activated. Go to Installation tab > Gripper to activate it and run the program again.", "Not activated", False, True, True)
  end
  rq_set_pos_spd_for(0, 255, 5, "2")
  rq_wait_pos_spe_for_request(0, 255, 5, "2")
  rq_go_to("2")
  rq_wait("2")
  # end: URCap Program Node
  $ 61 "'odpre prijemalo'"
  # 'odpre prijemalo'
  $ 62 "MoveL"
  $ 63 "Waypoint_01" "breakAfter"
  movel(Waypoint_01_p, a=1.2, v=0.25)
  $ 64 "'se umakne za potisk pokrova'"
  # 'se umakne za potisk pokrova'
  $ 65 "MoveL"
  $ 66 "Waypoint_001" "breakAfter"
  movel(Waypoint_001_p, a=1.2, v=0.25)
  $ 67 "'vmesen korak za potisk pokrova'"
  # 'vmesen korak za potisk pokrova'
  $ 68 "MoveL"
  $ 69 "Waypoint_02" "breakAfter"
  movel(Waypoint_02_p, a=1.2, v=0.25)
  $ 70 "'se pripravi za potisk pokrova'"
  # 'se pripravi za potisk pokrova'
  $ 71 "MoveL"
  $ 72 "Waypoint_03" "breakAfter"
  movel(Waypoint_03_p, a=1.2, v=0.25)
  $ 73 "'potisne pokrov'"
  # 'potisne pokrov'
  $ 74 "MoveL"
  $ 75 "Waypoint_11" "breakAfter"
  movel(Waypoint_11_p, a=1.2, v=0.25)
  $ 76 "'stran od skatle'"
  # 'stran od skatle'
  $ 77 "Waypoint_13" "breakAfter"
  movel(Waypoint_13_p, a=1.2, v=0.25)
  $ 78 "'domov = opravi task'"
  # 'domov = opravi task'
  $ 79 "Wait: 2.0"
  sleep(2.0)
  $ 80 "Waypoint_11" "breakAfter"
  movel(Waypoint_11_p, a=1.2, v=0.25)
  $ 81 "'se postavi nad skatlo'"
  # 'se postavi nad skatlo'
  # begin: URCap Program Node
  #   Source: Robotiq_Grippers, 1.8.3.4198-beta, Robotiq Inc.
  #   Type: Gripper
  $ 82 "Gripper Open (2)"
  if not(gripper_connected[1]):
    popup("Gripper 2 must be connected to run this program.", "No connection", False, True, True)
  end
  if not(rq_is_gripper_activated("2")):
    popup("Gripper 2 is not activated. Go to Installation tab > Gripper to activate it and run the program again.", "Not activated", False, True, True)
  end
  rq_set_pos_spd_for(0, 255, 5, "2")
  rq_wait_pos_spe_for_request(0, 255, 5, "2")
  rq_go_to("2")
  rq_wait("2")
  # end: URCap Program Node
  $ 83 "'odpre gripper'"
  # 'odpre gripper'
  $ 84 "Waypoint_04" "breakAfter"
  movel(Waypoint_04_p, a=1.2, v=0.25)
  $ 85 "'premik nad pozicijo za pobiranje pokrova'"
  # 'premik nad pozicijo za pobiranje pokrova'
  $ 86 "Waypoint_05" "breakAfter"
  movel(Waypoint_05_p, a=1.2, v=0.25)
  $ 87 "'premik na pozicijo za pobiranje pokrova'"
  # 'premik na pozicijo za pobiranje pokrova'
  # begin: URCap Program Node
  #   Source: Robotiq_Grippers, 1.8.3.4198-beta, Robotiq Inc.
  #   Type: Gripper
  $ 88 "Gripper Close (2)"
  if not(gripper_connected[1]):
    popup("Gripper 2 must be connected to run this program.", "No connection", False, True, True)
  end
  if not(rq_is_gripper_activated("2")):
    popup("Gripper 2 is not activated. Go to Installation tab > Gripper to activate it and run the program again.", "Not activated", False, True, True)
  end
  rq_set_pos_spd_for(255, 255, 77, "2")
  rq_wait_pos_spe_for_request(255, 255, 77, "2")
  rq_go_to("2")
  rq_wait("2")
  # end: URCap Program Node
  $ 89 "'zapre prijemalo'"
  # 'zapre prijemalo'
  $ 90 "Waypoint_06" "breakAfter"
  movel(Waypoint_06_p, a=1.2, v=0.25)
  $ 91 "'dvigne pokrov'"
  # 'dvigne pokrov'
  $ 92 "Waypoint_14" "breakAfter"
  movel(Waypoint_14_p, a=1.2, v=0.25)
  $ 93 "'pokrov postavi v zacetno pozicijo'"
  # 'pokrov postavi v zacetno pozicijo'
  $ 94 "If open_socket"
  if (open_socket):
    $ 95 "was_send≔socket_send_string('ZAPRTA','student')"
    global was_send=socket_send_string("ZAPRTA","student")
    $ 96 "Loop  not was_send"
    while (  not  was_send):
      $ 97 "was_send≔socket_send_string('ZAPRTA','student')"
      global was_send=socket_send_string("ZAPRTA","student")
      $ 98 "Wait: 0.01"
      sleep(0.01)
    end
    $ 99 "Wait: 0.01"
    sleep(0.01)
  end
  # begin: URCap Program Node
  #   Source: Robotiq_Grippers, 1.8.3.4198-beta, Robotiq Inc.
  #   Type: Gripper
  $ 100 "Gripper Open (2)"
  if not(gripper_connected[1]):
    popup("Gripper 2 must be connected to run this program.", "No connection", False, True, True)
  end
  if not(rq_is_gripper_activated("2")):
    popup("Gripper 2 is not activated. Go to Installation tab > Gripper to activate it and run the program again.", "Not activated", False, True, True)
  end
  rq_set_pos_spd_for(0, 255, 5, "2")
  rq_wait_pos_spe_for_request(0, 255, 5, "2")
  rq_go_to("2")
  rq_wait("2")
  # end: URCap Program Node
  $ 101 "'odpre gripper'"
  # 'odpre gripper'
  $ 102 "Set DO[0]=On"
  set_standard_digital_out(0, True)
  $ 103 "'vklopi napajanje za kljucavnico'"
  # 'vklopi napajanje za kljucavnico'
  $ 104 "Wait: 1.0"
  sleep(1.0)
  $ 105 "Set DO[0]=Off"
  set_standard_digital_out(0, False)
  $ 106 "'izklopi napajanje za kljucavnico'"
  # 'izklopi napajanje za kljucavnico'
  $ 107 "If open_socket"
  if (open_socket):
    $ 108 "was_send≔socket_send_string('ZAKLENJENA','student')"
    global was_send=socket_send_string("ZAKLENJENA","student")
    $ 109 "Loop  not was_send"
    while (  not  was_send):
      $ 110 "was_send≔socket_send_string('ZAKLENJENA','student')"
      global was_send=socket_send_string("ZAKLENJENA","student")
      $ 111 "Wait: 0.01"
      sleep(0.01)
    end
    $ 112 "Wait: 0.01"
    sleep(0.01)
  end
  $ 113 "Waypoint_13" "breakAfter"
  movel(Waypoint_13_p, a=1.2, v=0.25)
  $ 114 "'domov'"
  # 'domov'
  $ 115 "If digital_in[5]"
  if (get_standard_digital_in(5)):
    $ 116 "Set DO[5]=On"
    set_standard_digital_out(5, True)
    $ 117 "'ce je skatla se pri senzorju posljemo naprej'"
    # 'ce je skatla se pri senzorju posljemo naprej'
    $ 118 "'tcp_ip skatla sla naprej'"
    # 'tcp_ip skatla sla naprej'
    $ 119 "If open_socket"
    if (open_socket):
      $ 120 "was_send≔socket_send_string('ODPRAVLJENA','student')"
      global was_send=socket_send_string("ODPRAVLJENA","student")
      $ 121 "Loop  not was_send"
      while (  not  was_send):
        $ 122 "was_send≔socket_send_string('ODPRAVLJENA','student')"
        global was_send=socket_send_string("ODPRAVLJENA","student")
        $ 123 "Wait: 0.01"
        sleep(0.01)
      end
      $ 124 "Wait: 0.01"
      sleep(0.01)
    end
  end
  $ 125 "Loop digital_in[5]"
  while (get_standard_digital_in(5)):
    $ 126 "'cakam da skatla ne bo vec pri senzorju'"
    # 'cakam da skatla ne bo vec pri senzorju'
  end
  $ 127 "Set DO[5]=Off"
  set_standard_digital_out(5, False)
  $ 128 "socket_close('student')"
  socket_close("student")
  $ 129 "Halt"
  halt
end
